// TIA Portal V17 export
// export: Created 2022-07-20T06:59:50.9223884Z, ExportSetting WithDefaults, DisplayName Totally Integrated Automation Portal, DisplayVersion V17, DisplayName TIA Portal Openness, DisplayVersion V17, DisplayName TIA Portal Version Control Interface, DisplayVersion V17, DisplayName SINAMICS Startdrive Advanced, DisplayVersion V17, DisplayName SINAMICS Startdrive G130, G150, S120, S150, SINAMICS MV, S210, DisplayVersion V17, DisplayName SINAMICS Startdrive G110M, G120, G120C, G120D, G120P, G115D, DisplayVersion V17, DisplayName STEP 7 Professional, DisplayVersion V17, DisplayName STEP 7 Safety, DisplayVersion V17, DisplayName WinCC Advanced, DisplayVersion V17
FUNCTION_BLOCK "FB10063_IperCleaningInkCircuit"   // FB10063, LAD
{ S7_Optimized_Access := 'TRUE' }
VERSION : 0.1
// stored: AutoNumber false, IsIECCheckEnabled false, IsRetainMemResEnabled false, MemoryReserve 100, SetENOAutomatically false, UDAEnableTagReadback false
   VAR_INPUT
      PipeFlushSensor : Bool;
      FlushInWeighScale_RawWeight : Int;
      FlushInWeighScale_CalibrationWeight_1 : Real;
      FlushInWeighScale_CalibrationWeight_2 : Real;
      FlushInWeighScale_LowWarningThreshold : Real;
      FlushInWeighScale_HighWarningThreshold : Real;
      FlushInWeighScale_LowErrorThreshold : Real;
      FlushInWeighScale_HighErrorThreshold : Real;
      FlushOutWeighScale_RawValue : Int;
      FlushOutWeighScale_CalibrationWeight_1 : Real;
      FlushOutWeighScale_CalibrationWeight_2 : Real;
      FlushOutWeighScale_LowWarningThreshold : Real;
      FlushOutWeighScale_HighWarningThreshold : Real;
      FlushOutWeighScale_LowErrorThreshold : Real;
      FlushOutWeighScale_HighErrorThreshold : Real;
      FlushWasteWeighScale_RawValue : Int;
      FlushWasteWeighScale_CalibrationWeight_1 : Real;
      FlushWasteWeighScale_CalibrationWeight_2 : Real;
      FlushWasteWeighScale_LowWarningThreshold : Real;
      FlushWasteWeighScale_HighWarningThreshold : Real;
      FlushWasteWeighScale_LowErrorThreshold : Real;
      FlushWasteWeighScale_HighErrorThreshold : Real;
      FillCappingStationTime : Time := T#70s;
      DrainCappingStationTime : Time := T#120s;
   END_VAR
   VAR_OUTPUT
      ActiveFlushInPump : Bool;
      ActiveFlushInSolenoidValve : Bool;
      ActiveFlushOutPump : Bool;
      ActiveFlushOutSolenoidValve : Bool;
      ActiveFlushWastePump : Bool;
      ActiveFlushWasteSolenoidValve : Bool;
      FlushInWeighScale_CalibrationStatus_1 : Bool;
      FlushInWeighScale_CalibrationStatus_2 : Bool;
      FlushInWeighScale_LowWarningThresholdReached : Bool;
      FlushInWeighScale_HighWarningThresholdReached : Bool;
      FlushInWeighScale_LowErrorThresholdReached : Bool;
      FlushInWeighScale_HighErrorThresholdReached : Bool;
      FlushInWeighScale_ActualValue : Real;
      "FlushInWeighScale_ActualValue_%" : Real;
      FlushInWeighScale_SensorCalibrated : Bool;
      FlushOutWeighScale_CalibrationStatus_1 : Bool;
      FlushOutWeighScale_CalibrationStatus_2 : Bool;
      FlushOutWeighScale_LowWarningThresholdReached : Bool;
      FlushOutWeighScale_HighWarningThresholdReached : Bool;
      FlushOutWeighScale_LowErrorThresholdReached : Bool;
      FlushOutWeighScale_HighErrorThresholdReached : Bool;
      FlushOutWeighScale_ActualValue : Real;
      "FlushOutWeighScale_ActualValue_%" : Real;
      FlushOutWeighScale_SensorCalibrated : Bool;
      FlushWasteWeighScale_CalibrationStatus_1 : Bool;
      FlushWasteWeighScale_CalibrationStatus_2 : Bool;
      FlushWasteWeighScale_LowWarningThresholdReached : Bool;
      FlushWasteWeighScale_HighWarningThresholdReached : Bool;
      FlushWasteWeighScale_LowErrorThresholdReached : Bool;
      FlushWasteWeighScale_HighErrorThresholdReached : Bool;
      FlushWasteWeighScale_ActualValue : Real;
      "FlushWasteWeighScale_ActualValue_%" : Real;
      FlushWasteWeighScale_SensorCalibrated : Bool;
      FillCappingStationInProgress : Bool;
      FillCappingStationDone : Bool;
      DrainCappingStationInProgress : Bool;
      DrainCappingStationDone : Bool;
      CleaningInkCircuitInError : Bool;
   END_VAR
   VAR_IN_OUT
      RequestFillCappingStation : Bool;
      RequestDrainCappingStation : Bool;
      RequestDrainFlushWaste : Bool;
      FlushInWeighScale_CalibrationDataX_1 : Real;
      FlushInWeighScale_CalibrationDataY_1 : Real;
      FlushInWeighScale_CalibrationDataX_2 : Real;
      FlushInWeighScale_RequestCalibration_1 : Bool;
      FlushInWeighScale_ResetCalibration : Bool;
      FlushInWeighScale_RequestCalibration_2 : Bool;
      FlushInWeighScale_CalibrationDataY_2 : Real;
      FlushOutWeighScale_CalibrationDataX_1 : Real;
      FlushOutWeighScale_CalibrationDataY_1 : Real;
      FlushOutWeighScale_CalibrationDataX_2 : Real;
      FlushOutWeighScale_CalibrationDataY_2 : Real;
      FlushOutWeighScale_RequestCalibration_1 : Bool;
      FlushOutWeighScale_ResetCalibration : Bool;
      FlushOutWeighScale_RequestCalibration_2 : Bool;
      FlushWasteWeighScale_CalibrationDataX_1 : Real;
      FlushWasteWeighScale_CalibrationDataY_1 : Real;
      FlushWasteWeighScale_CalibrationDataX_2 : Real;
      FlushWasteWeighScale_CalibrationDataY_2 : Real;
      FlushWasteWeighScale_RequestCalibration_1 : Bool;
      FlushWasteWeighScale_RequestCalibration_2 : Bool;
      FlushWasteWeighScale_ResetCalibration : Bool;
   END_VAR
   VAR
      CappingStationManagementStateDiagram : Int;
      FlushWasteManagementStateDiagram : Int;
      R_TRIG_RequestFillFlushPipe : R_TRIG;
      R_TRIG_RequestFillCappingStation : R_TRIG;
      R_TRIG_RequestDrainCappingStation : R_TRIG;
      R_TRIG_RequestDrainFlushWaste { S7_SetPoint := 'True'} : R_TRIG;
      F_TRIG_RequestFillCappingStation : F_TRIG;
      F_TRIG_RequestDrainCappingStation { S7_SetPoint := 'True'} : F_TRIG;
      F_TRIG_RequestDrainFlushWaste { S7_SetPoint := 'True'} : F_TRIG;
      TON_FIllCappingStationRecirculation { S7_SetPoint := 'True'} : TON_TIME;
      TON_FillCappingStation { S7_SetPoint := 'True'} : TON_TIME;
      TON_DrainCappingStationPipeSensor { S7_SetPoint := 'True'} : TON_TIME;
      TON_DrainCappingStation { S7_SetPoint := 'True'} : TON_TIME;
      TON_DrainFlushWasteCleaningTray { S7_SetPoint := 'True'} : TON_TIME;
      FB10030_AnalogicalSensor_TLMScale_FlushInWeighScale { S7_SetPoint := 'True'} : "FB10030_AnalogicalSensor";
      FB10030_AnalogicalSensor_TLMScale_FlushOutWeighScale { S7_SetPoint := 'True'} : "FB10030_AnalogicalSensor";
      FB10030_AnalogicalSensor_TLMScale_FlushWasteWeighScale { S7_SetPoint := 'True'} : "FB10030_AnalogicalSensor";
   END_VAR
   VAR CONSTANT
      WAIT_FOR_CAPPING_STATION_REQUEST : Int := 0;
      FILL_CAPPING_STATION_RECIRCULATION : Int := 10;
      FILL_CAPPING_STATION : Int := 20;
      DRAIN_CAPPING_STATION_PIPE_SENSOR : Int := 30;
      DRAIN_CAPPING_STATION : Int := 40;
      CLEANING_INK_REQUESTS_DONE : Int := 50;
      "==========" : Bool;
      WAIT_FOR_FLUSH_WASTE_REQUEST : Int := 0;
      DRAIN_FLUSH_WASTE_IN_PROGRESS : Int := 10;
      FLUSH_WASTE_REQUEST_DONE : Int := 20;
   END_VAR
BEGIN

REGION Network 1 (SCL): First Scan
   IF "FirstScan" THEN
       #FillCappingStationDone := FALSE;
       #DrainCappingStationDone := FALSE;

       #CappingStationManagementStateDiagram := #WAIT_FOR_CAPPING_STATION_REQUEST;
       #FlushWasteManagementStateDiagram := #WAIT_FOR_FLUSH_WASTE_REQUEST;
   END_IF;
END_REGION

REGION Network 2 (SCL): Edge Signals & Timers
   REGION EDGE SIGNALS
       #R_TRIG_RequestFillCappingStation(CLK := #RequestFillCappingStation);
       #R_TRIG_RequestDrainCappingStation(CLK := #RequestDrainCappingStation);
       #R_TRIG_RequestDrainFlushWaste(CLK := #RequestDrainFlushWaste);

       #F_TRIG_RequestFillCappingStation(CLK := #RequestFillCappingStation);
       #F_TRIG_RequestDrainCappingStation(CLK := #RequestDrainCappingStation);
       #F_TRIG_RequestDrainFlushWaste(CLK := #RequestDrainFlushWaste);
   END_REGION

   REGION TIMERS
       #TON_FIllCappingStationRecirculation(IN := #PipeFlushSensor AND #CappingStationManagementStateDiagram = #FILL_CAPPING_STATION_RECIRCULATION,
                                           PT := T#5s);
       #TON_FillCappingStation(IN := #CappingStationManagementStateDiagram = #FILL_CAPPING_STATION,
                               PT := #FillCappingStationTime);
       #TON_DrainCappingStationPipeSensor(IN := NOT (#PipeFlushSensor) AND #CappingStationManagementStateDiagram = #DRAIN_CAPPING_STATION_PIPE_SENSOR,
                                          PT := T#5s);
       #TON_DrainCappingStation(IN := #CappingStationManagementStateDiagram = #DRAIN_CAPPING_STATION,
                                PT := #DrainCappingStationTime);
       #TON_DrainFlushWasteCleaningTray(IN := #FlushWasteManagementStateDiagram = #DRAIN_FLUSH_WASTE_IN_PROGRESS,
                                        PT := T#30s);
   END_REGION
END_REGION

REGION Network 3: Flush In Weigh Scale Management
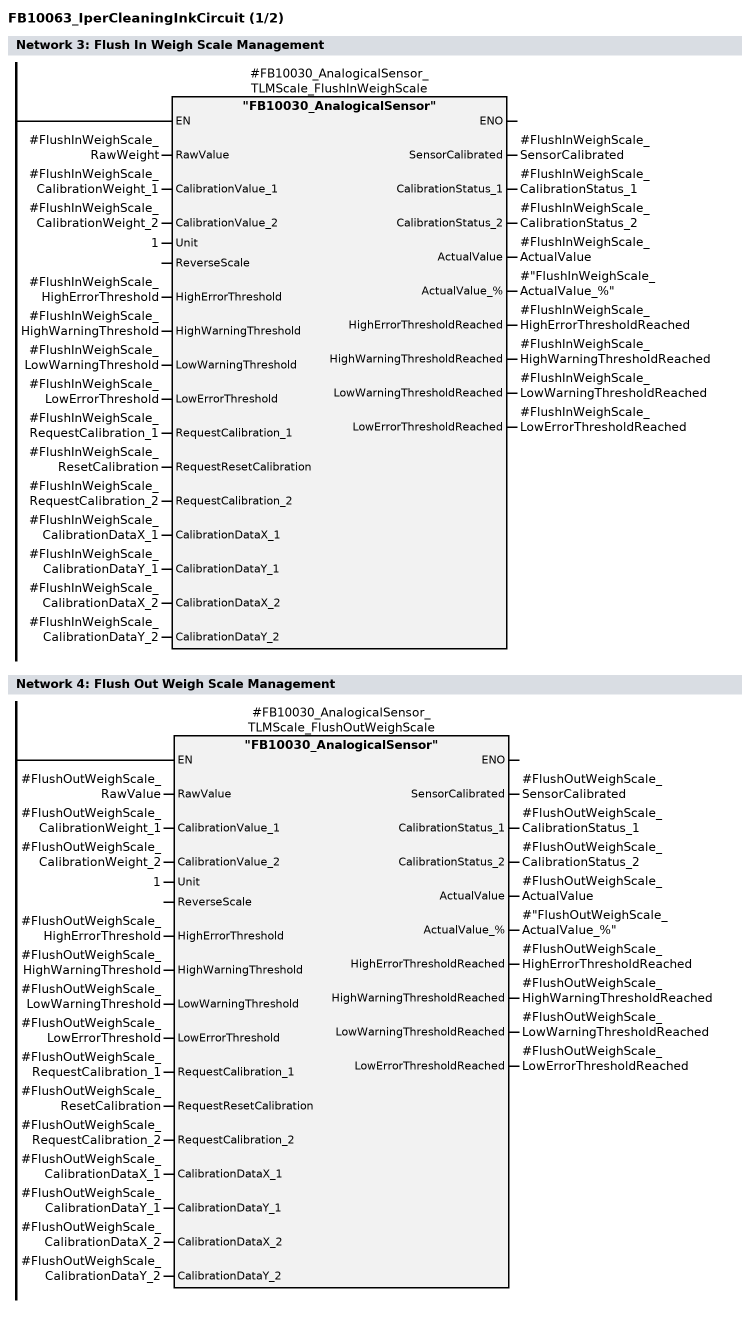
   RUNG wire#powerrail
      #FB10030_AnalogicalSensor_TLMScale_FlushInWeighScale(RawValue := #FlushInWeighScale_RawWeight, CalibrationValue_1 := #FlushInWeighScale_CalibrationWeight_1, CalibrationValue_2 := #FlushInWeighScale_CalibrationWeight_2, Unit := 1, ReverseScale :=, HighErrorThreshold := #FlushInWeighScale_HighErrorThreshold, HighWarningThreshold := #FlushInWeighScale_HighWarningThreshold, LowWarningThreshold := #FlushInWeighScale_LowWarningThreshold, LowErrorThreshold := #FlushInWeighScale_LowErrorThreshold, RequestCalibration_1 := #FlushInWeighScale_RequestCalibration_1, RequestCalibration_2 := #FlushInWeighScale_RequestCalibration_2, RequestResetCalibration := #FlushInWeighScale_ResetCalibration, CalibrationDataX_1 := #FlushInWeighScale_CalibrationDataX_1, CalibrationDataY_1 := #FlushInWeighScale_CalibrationDataY_1, CalibrationDataX_2 := #FlushInWeighScale_CalibrationDataX_2, CalibrationDataY_2 := #FlushInWeighScale_CalibrationDataY_2, SensorCalibrated => #FlushInWeighScale_SensorCalibrated, CalibrationStatus_1 => #FlushInWeighScale_CalibrationStatus_1, CalibrationStatus_2 => #FlushInWeighScale_CalibrationStatus_2, ActualValue => #FlushInWeighScale_ActualValue, "ActualValue_%" => #"FlushInWeighScale_ActualValue_%", HighErrorThresholdReached => #FlushInWeighScale_HighErrorThresholdReached, HighWarningThresholdReached => #FlushInWeighScale_HighWarningThresholdReached, LowWarningThresholdReached => #FlushInWeighScale_LowWarningThresholdReached, LowErrorThresholdReached => #FlushInWeighScale_LowErrorThresholdReached)
   END_RUNG
   // the same network as SCL:
   #FB10030_AnalogicalSensor_TLMScale_FlushInWeighScale(RawValue := #FlushInWeighScale_RawWeight,   // "FB10030_AnalogicalSensor"
                           CalibrationValue_1 := #FlushInWeighScale_CalibrationWeight_1,
                           CalibrationValue_2 := #FlushInWeighScale_CalibrationWeight_2,
                           Unit := 1,
                           HighErrorThreshold := #FlushInWeighScale_HighErrorThreshold,
                           HighWarningThreshold := #FlushInWeighScale_HighWarningThreshold,
                           LowWarningThreshold := #FlushInWeighScale_LowWarningThreshold,
                           LowErrorThreshold := #FlushInWeighScale_LowErrorThreshold,
                           RequestCalibration_1 := #FlushInWeighScale_RequestCalibration_1,
                           RequestResetCalibration := #FlushInWeighScale_ResetCalibration,
                           RequestCalibration_2 := #FlushInWeighScale_RequestCalibration_2,
                           CalibrationDataX_1 := #FlushInWeighScale_CalibrationDataX_1,
                           CalibrationDataY_1 := #FlushInWeighScale_CalibrationDataY_1,
                           CalibrationDataX_2 := #FlushInWeighScale_CalibrationDataX_2,
                           CalibrationDataY_2 := #FlushInWeighScale_CalibrationDataY_2,
                           SensorCalibrated => #FlushInWeighScale_SensorCalibrated,
                           CalibrationStatus_1 => #FlushInWeighScale_CalibrationStatus_1,
                           CalibrationStatus_2 => #FlushInWeighScale_CalibrationStatus_2,
                           ActualValue => #FlushInWeighScale_ActualValue,
                           "ActualValue_%" => #"FlushInWeighScale_ActualValue_%",
                           HighErrorThresholdReached => #FlushInWeighScale_HighErrorThresholdReached,
                           HighWarningThresholdReached => #FlushInWeighScale_HighWarningThresholdReached,
                           LowWarningThresholdReached => #FlushInWeighScale_LowWarningThresholdReached,
                           LowErrorThresholdReached => #FlushInWeighScale_LowErrorThresholdReached);
END_REGION

REGION Network 4: Flush Out Weigh Scale Management
   RUNG wire#powerrail
      #FB10030_AnalogicalSensor_TLMScale_FlushOutWeighScale(RawValue := #FlushOutWeighScale_RawValue, CalibrationValue_1 := #FlushOutWeighScale_CalibrationWeight_1, CalibrationValue_2 := #FlushOutWeighScale_CalibrationWeight_2, Unit := 1, ReverseScale :=, HighErrorThreshold := #FlushOutWeighScale_HighErrorThreshold, HighWarningThreshold := #FlushOutWeighScale_HighWarningThreshold, LowWarningThreshold := #FlushOutWeighScale_LowWarningThreshold, LowErrorThreshold := #FlushOutWeighScale_LowErrorThreshold, RequestCalibration_1 := #FlushOutWeighScale_RequestCalibration_1, RequestResetCalibration := #FlushOutWeighScale_ResetCalibration, RequestCalibration_2 := #FlushOutWeighScale_RequestCalibration_2, CalibrationDataX_1 := #FlushOutWeighScale_CalibrationDataX_1, CalibrationDataY_1 := #FlushOutWeighScale_CalibrationDataY_1, CalibrationDataX_2 := #FlushOutWeighScale_CalibrationDataX_2, CalibrationDataY_2 := #FlushOutWeighScale_CalibrationDataY_2, SensorCalibrated => #FlushOutWeighScale_SensorCalibrated, CalibrationStatus_1 => #FlushOutWeighScale_CalibrationStatus_1, CalibrationStatus_2 => #FlushOutWeighScale_CalibrationStatus_2, ActualValue => #FlushOutWeighScale_ActualValue, "ActualValue_%" => #"FlushOutWeighScale_ActualValue_%", HighErrorThresholdReached => #FlushOutWeighScale_HighErrorThresholdReached, HighWarningThresholdReached => #FlushOutWeighScale_HighWarningThresholdReached, LowWarningThresholdReached => #FlushOutWeighScale_LowWarningThresholdReached, LowErrorThresholdReached => #FlushOutWeighScale_LowErrorThresholdReached)
   END_RUNG
   // the same network as SCL:
   #FB10030_AnalogicalSensor_TLMScale_FlushOutWeighScale(RawValue := #FlushOutWeighScale_RawValue,   // "FB10030_AnalogicalSensor"
                           CalibrationValue_1 := #FlushOutWeighScale_CalibrationWeight_1,
                           CalibrationValue_2 := #FlushOutWeighScale_CalibrationWeight_2,
                           Unit := 1,
                           HighErrorThreshold := #FlushOutWeighScale_HighErrorThreshold,
                           HighWarningThreshold := #FlushOutWeighScale_HighWarningThreshold,
                           LowWarningThreshold := #FlushOutWeighScale_LowWarningThreshold,
                           LowErrorThreshold := #FlushOutWeighScale_LowErrorThreshold,
                           RequestCalibration_1 := #FlushOutWeighScale_RequestCalibration_1,
                           RequestResetCalibration := #FlushOutWeighScale_ResetCalibration,
                           RequestCalibration_2 := #FlushOutWeighScale_RequestCalibration_2,
                           CalibrationDataX_1 := #FlushOutWeighScale_CalibrationDataX_1,
                           CalibrationDataY_1 := #FlushOutWeighScale_CalibrationDataY_1,
                           CalibrationDataX_2 := #FlushOutWeighScale_CalibrationDataX_2,
                           CalibrationDataY_2 := #FlushOutWeighScale_CalibrationDataY_2,
                           SensorCalibrated => #FlushOutWeighScale_SensorCalibrated,
                           CalibrationStatus_1 => #FlushOutWeighScale_CalibrationStatus_1,
                           CalibrationStatus_2 => #FlushOutWeighScale_CalibrationStatus_2,
                           ActualValue => #FlushOutWeighScale_ActualValue,
                           "ActualValue_%" => #"FlushOutWeighScale_ActualValue_%",
                           HighErrorThresholdReached => #FlushOutWeighScale_HighErrorThresholdReached,
                           HighWarningThresholdReached => #FlushOutWeighScale_HighWarningThresholdReached,
                           LowWarningThresholdReached => #FlushOutWeighScale_LowWarningThresholdReached,
                           LowErrorThresholdReached => #FlushOutWeighScale_LowErrorThresholdReached);
END_REGION

REGION Network 5: Flush Waste Weigh Scale Management
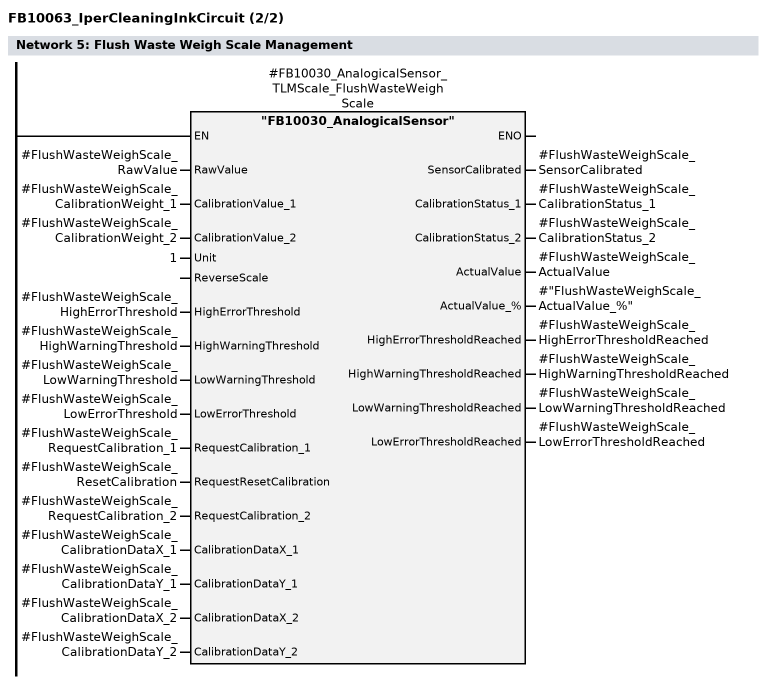
   RUNG wire#powerrail
      #FB10030_AnalogicalSensor_TLMScale_FlushWasteWeighScale(RawValue := #FlushWasteWeighScale_RawValue, CalibrationValue_1 := #FlushWasteWeighScale_CalibrationWeight_1, CalibrationValue_2 := #FlushWasteWeighScale_CalibrationWeight_2, Unit := 1, ReverseScale :=, HighErrorThreshold := #FlushWasteWeighScale_HighErrorThreshold, HighWarningThreshold := #FlushWasteWeighScale_HighWarningThreshold, LowWarningThreshold := #FlushWasteWeighScale_LowWarningThreshold, LowErrorThreshold := #FlushWasteWeighScale_LowErrorThreshold, RequestCalibration_1 := #FlushWasteWeighScale_RequestCalibration_1, RequestCalibration_2 := #FlushWasteWeighScale_RequestCalibration_2, RequestResetCalibration := #FlushWasteWeighScale_ResetCalibration, CalibrationDataX_1 := #FlushWasteWeighScale_CalibrationDataX_1, CalibrationDataY_1 := #FlushWasteWeighScale_CalibrationDataY_1, CalibrationDataX_2 := #FlushWasteWeighScale_CalibrationDataX_2, CalibrationDataY_2 := #FlushWasteWeighScale_CalibrationDataY_2, SensorCalibrated => #FlushWasteWeighScale_SensorCalibrated, CalibrationStatus_1 => #FlushWasteWeighScale_CalibrationStatus_1, CalibrationStatus_2 => #FlushWasteWeighScale_CalibrationStatus_2, ActualValue => #FlushWasteWeighScale_ActualValue, "ActualValue_%" => #"FlushWasteWeighScale_ActualValue_%", HighErrorThresholdReached => #FlushWasteWeighScale_HighErrorThresholdReached, HighWarningThresholdReached => #FlushWasteWeighScale_HighWarningThresholdReached, LowWarningThresholdReached => #FlushWasteWeighScale_LowWarningThresholdReached, LowErrorThresholdReached => #FlushWasteWeighScale_LowErrorThresholdReached)
   END_RUNG
   // the same network as SCL:
   #FB10030_AnalogicalSensor_TLMScale_FlushWasteWeighScale(RawValue := #FlushWasteWeighScale_RawValue,   // "FB10030_AnalogicalSensor"
                           CalibrationValue_1 := #FlushWasteWeighScale_CalibrationWeight_1,
                           CalibrationValue_2 := #FlushWasteWeighScale_CalibrationWeight_2,
                           Unit := 1,
                           HighErrorThreshold := #FlushWasteWeighScale_HighErrorThreshold,
                           HighWarningThreshold := #FlushWasteWeighScale_HighWarningThreshold,
                           LowWarningThreshold := #FlushWasteWeighScale_LowWarningThreshold,
                           LowErrorThreshold := #FlushWasteWeighScale_LowErrorThreshold,
                           RequestCalibration_1 := #FlushWasteWeighScale_RequestCalibration_1,
                           RequestResetCalibration := #FlushWasteWeighScale_ResetCalibration,
                           RequestCalibration_2 := #FlushWasteWeighScale_RequestCalibration_2,
                           CalibrationDataX_1 := #FlushWasteWeighScale_CalibrationDataX_1,
                           CalibrationDataY_1 := #FlushWasteWeighScale_CalibrationDataY_1,
                           CalibrationDataX_2 := #FlushWasteWeighScale_CalibrationDataX_2,
                           CalibrationDataY_2 := #FlushWasteWeighScale_CalibrationDataY_2,
                           SensorCalibrated => #FlushWasteWeighScale_SensorCalibrated,
                           CalibrationStatus_1 => #FlushWasteWeighScale_CalibrationStatus_1,
                           CalibrationStatus_2 => #FlushWasteWeighScale_CalibrationStatus_2,
                           ActualValue => #FlushWasteWeighScale_ActualValue,
                           "ActualValue_%" => #"FlushWasteWeighScale_ActualValue_%",
                           HighErrorThresholdReached => #FlushWasteWeighScale_HighErrorThresholdReached,
                           HighWarningThresholdReached => #FlushWasteWeighScale_HighWarningThresholdReached,
                           LowWarningThresholdReached => #FlushWasteWeighScale_LowWarningThresholdReached,
                           LowErrorThresholdReached => #FlushWasteWeighScale_LowErrorThresholdReached);
END_REGION

REGION Network 6 (SCL): Cleaning Ink Circuit Management
   REGION CAPPING STATION MANAGEMENT
       CASE #CappingStationManagementStateDiagram OF
           #WAIT_FOR_CAPPING_STATION_REQUEST:
               IF #R_TRIG_RequestFillCappingStation.Q THEN
                   #FillCappingStationDone := FALSE;
                   #CappingStationManagementStateDiagram := #FILL_CAPPING_STATION_RECIRCULATION;
               ELSIF #R_TRIG_RequestDrainCappingStation.Q THEN
                   #DrainCappingStationDone := FALSE;
                   #CappingStationManagementStateDiagram := #DRAIN_CAPPING_STATION_PIPE_SENSOR;
               END_IF;
           #FILL_CAPPING_STATION_RECIRCULATION:
               #ActiveFlushInPump := TRUE;
               #ActiveFlushInSolenoidValve := TRUE;
               #ActiveFlushOutPump := TRUE;
               #ActiveFlushOutSolenoidValve := TRUE;
               #FillCappingStationInProgress := TRUE;
               IF #TON_FIllCappingStationRecirculation.Q THEN
                   #ActiveFlushOutPump := FALSE;
                   #ActiveFlushOutSolenoidValve := FALSE;
                   #CappingStationManagementStateDiagram := #FILL_CAPPING_STATION;
               ELSIF #F_TRIG_RequestFillCappingStation.Q THEN
                   #ActiveFlushInPump := FALSE;
                   #ActiveFlushInSolenoidValve := FALSE;
                   #ActiveFlushOutPump := FALSE;
                   #ActiveFlushOutSolenoidValve := FALSE;
                   #FillCappingStationInProgress := FALSE;
                   #CappingStationManagementStateDiagram := #CLEANING_INK_REQUESTS_DONE;
               END_IF;
           #FILL_CAPPING_STATION:
               #ActiveFlushInSolenoidValve := TRUE;
               #ActiveFlushInPump := TRUE;
               IF #TON_FillCappingStation.Q OR #F_TRIG_RequestFillCappingStation.Q THEN
                   #ActiveFlushInSolenoidValve := FALSE;
                   #ActiveFlushInPump := FALSE;
                   #FillCappingStationInProgress := FALSE;
                   #FillCappingStationDone := TRUE;
                   #CappingStationManagementStateDiagram := #CLEANING_INK_REQUESTS_DONE;
               END_IF;
           #DRAIN_CAPPING_STATION:
               #ActiveFlushOutSolenoidValve := TRUE;
               #ActiveFlushOutPump := TRUE;
               #DrainCappingStationInProgress := TRUE;
               IF #TON_DrainCappingStationPipeSensor.Q THEN
                   #ActiveFlushOutSolenoidValve := FALSE;
                   #ActiveFlushOutPump := FALSE;
                   #DrainCappingStationInProgress := FALSE;
                   #CappingStationManagementStateDiagram := #CLEANING_INK_REQUESTS_DONE;
               ELSIF #F_TRIG_RequestDrainCappingStation.Q THEN
                   #ActiveFlushOutSolenoidValve := FALSE;
                   #ActiveFlushOutPump := FALSE;
                   #CappingStationManagementStateDiagram := #DRAIN_CAPPING_STATION_PIPE_SENSOR;
               END_IF;
           #DRAIN_CAPPING_STATION_PIPE_SENSOR:
               #ActiveFlushOutSolenoidValve := TRUE;
               #ActiveFlushOutPump := TRUE;
               IF #TON_DrainCappingStation.Q OR #F_TRIG_RequestDrainCappingStation.Q THEN
                   #ActiveFlushOutSolenoidValve := FALSE;
                   #ActiveFlushOutPump := FALSE;
                   #DrainCappingStationDone := TRUE;
                   #DrainCappingStationInProgress := FALSE;
                   #CappingStationManagementStateDiagram := #CLEANING_INK_REQUESTS_DONE;
               END_IF;
           #CLEANING_INK_REQUESTS_DONE:
               #CappingStationManagementStateDiagram := #WAIT_FOR_CAPPING_STATION_REQUEST;
       END_CASE;
   END_REGION

   REGION FLUSH WASTE MANAGEMENT
       CASE #FlushWasteManagementStateDiagram OF
           #WAIT_FOR_FLUSH_WASTE_REQUEST:
               IF #R_TRIG_RequestDrainFlushWaste.Q THEN
                   #FlushWasteManagementStateDiagram := #DRAIN_FLUSH_WASTE_IN_PROGRESS;
               END_IF;
           #DRAIN_FLUSH_WASTE_IN_PROGRESS:
               //Request For Flush Waste Circuit
               #ActiveFlushWastePump := TRUE;
               #ActiveFlushWasteSolenoidValve := TRUE;

               //Condition To Go To Next Step
               IF #TON_DrainFlushWasteCleaningTray.Q OR #F_TRIG_RequestDrainFlushWaste.Q THEN
                   #ActiveFlushWastePump := FALSE;
                   #ActiveFlushWasteSolenoidValve := FALSE;

                   #FlushWasteManagementStateDiagram := #FLUSH_WASTE_REQUEST_DONE;
               END_IF;
           #FLUSH_WASTE_REQUEST_DONE:
               #ActiveFlushWastePump := FALSE;
               #ActiveFlushWasteSolenoidValve := FALSE;

               #FlushWasteManagementStateDiagram := #FLUSH_WASTE_REQUEST_DONE;
       END_CASE;
   END_REGION
END_REGION
END_FUNCTION_BLOCK
